FUNCTION F_NN : ARRAY[0..0] OF LREAL;
VAR_INPUT
	input: ARRAY[0..1] OF LREAL;
END_VAR
VAR
	layers : Layers;
	layer_output : ARRAY[0..130] OF LREAL;
	layer_input : ARRAY[0..130] OF LREAL;
	i : UINT;
END_VAR

MEMCPY(destAddr:=ADR(layer_input),srcAddr:=ADR(input),n:=SIZEOF(input));
FOR i := 0 TO layers.num_layers-2 DO
	F_ForwardPropagation(	layer_pre	:= 	layers.layers[i],
							layer_next	:=	layers.layers[i+1],
							pointer_in 	:=	ADR(layer_input),
							pointer_out	:=	ADR(layer_output));
	MEMCPY(destAddr:=ADR(layer_input),srcAddr:=ADR(layer_output),n:=SIZEOF(LREAL)*layers.layers[i+1].num_neurons);
END_FOR
MEMCPY(destAddr:=ADR(F_NN),srcAddr:=ADR(layer_output),n:=SIZEOF(F_NN));

END_FUNCTION

(* stored: Version 1.1.0.1, ProductVersion 3.1.4024.12
   POU F_NN: Id {07ce18b5-fe38-4fc1-8aea-e0a271c85924}, SpecialFunc None *)
